{attribute 'qualified_only'}
{attribute 'strict'}
TYPE EBoolOperation :
(
	none := 0,
	and_op := 1,
	nand_op := 2,
	or_op := 3,
	nor_op := 4
);
END_TYPE

(* stored: Version 1.1.0.1, ProductVersion 3.1.4024.9
   DUT EBoolOperation: Id {858be62a-36a2-4d9c-b6f5-996ac1d7d401} *)
